PROGRAM MAIN
VAR
	dummyRunner : ObjectRunner;
	XtsRunnerTestSuite : XtsRunnerTesting;
//	XtsHardwareTestSuite : XtsHardwareTesting(dummyRunner);
END_VAR

XtsRunnerTestSuite();

END_PROGRAM

(* stored: Version 1.1.0.1, ProductVersion 3.1.4024.12
   POU MAIN: Id {aa92f88a-2917-437b-b76e-fd83d614eadb}, SpecialFunc None *)
